(* IEC 61131-3 sources: Industry-PLC-LLM/data/PLCBEAD_repo/PLCBEAD_PLCEmbed-main/PLC-BEAD/Source/GEB/SETUP_CHARNAMES, 1 file *)

(* ---- SETUP_CHARNAMES.ST ---- *)
TYPE
  oscat_CHARNAMES	: ARRAY [1..11] OF STRING;
END_TYPE

FUNCTION_BLOCK SETUP_CHARNAMES_Block

	VAR_IN_OUT
		CHARNAMES :	oscat_CHARNAMES;
	END_VAR

	VAR
		init :	BOOL;
	END_VAR

	IF init THEN RETURN; END_IF;

	init := TRUE;

	CHARNAMES[01] := '123';
	CHARNAMES[02] := '456';
	CHARNAMES[03] := 'zgsdafasf';
	CHARNAMES[04] := 'sadfsdfa';
	CHARNAMES[05] := 'asdfdsafdfds';
	CHARNAMES[06] := 'sadfsdfsdf';
	CHARNAMES[07] := 'sfsfdfdddd';
	CHARNAMES[08] := 'dddddted';
	CHARNAMES[10] := 'wer';
	CHARNAMES[11] := 'werwer';

END_FUNCTION_BLOCK

PROGRAM program0

	VAR
		CHARNAMES :	oscat_CHARNAMES;
		func_block : SETUP_CHARNAMES_Block;
  	END_VAR
	func_block.CHARNAMES  :=CHARNAMES;
	func_block();
	CHARNAMES := func_block.CHARNAMES;

END_PROGRAM
